// TIA Portal V19 export
TYPE "LEXCHANGETRAY_typeScanner_par"
// stored: Access Published
   STRUCT
      laddr : HW_ANY;
      dataLength : UInt;
      startBit : DInt;
      disable : Bool;
      busyStatusBits_1 : Bool;
      completionStatusBits_1 : Bool;
      errorStatusBits_1 : Bool;
   END_STRUCT;
END_TYPE
